ABB RAPID module: FrameFieldProbe.mod

MODULE FrameFieldProbe
    ! CrossArm - frame field probe: see tools/make_frame_field_probe.py.
    PERS tooldata ffStylus:=[TRUE,[[0,0,150],[1,0,0,0]],[3,[0,0,50],[1,0,0,0],0,0,0]];
    PERS wobjdata ffPallet:=[FALSE,TRUE,"",[[1000,0,800],[0,0,1,0]],[[0,0,0],[1,0,0,0]]];
    PERS wobjdata ffNest1:=[FALSE,TRUE,"",[[1000,0,800],[0,0,1,0]],[[0,0,0],[1,0,0,0]]];
    PERS wobjdata ffNest2:=[FALSE,TRUE,"",[[1000,0,800],[0,0,1,0]],[[0,0,0],[1,0,0,0]]];
    PERS wobjdata ffNest3:=[FALSE,TRUE,"",[[1000,0,800],[0,0,1,0]],[[0,0,0],[1,0,0,0]]];
    PERS wobjdata ffNest4:=[FALSE,TRUE,"",[[1000,0,800],[0,0,1,0]],[[0,0,0],[1,0,0,0]]];
    PERS wobjdata ffNest5:=[FALSE,TRUE,"",[[1000,0,800],[0,0,1,0]],[[0,0,0],[1,0,0,0]]];
    PERS wobjdata ffNest6:=[FALSE,TRUE,"",[[1000,0,800],[0,0,1,0]],[[0,0,0],[1,0,0,0]]];
    PERS wobjdata ffNest7:=[FALSE,TRUE,"",[[1000,0,800],[0,0,1,0]],[[0,0,0],[1,0,0,0]]];
    PERS wobjdata ffNest8:=[FALSE,TRUE,"",[[1000,0,800],[0,0,1,0]],[[30,0,0],[1,0,0,0]]];
    PERS wobjdata ffNest9:=[FALSE,TRUE,"",[[1000,0,800],[0,0,1,0]],[[0,20,0],[0.9659258,0,0,0.258819]]];
    CONST robtarget ffT1:=[[950,-60,820],[0,-0.1736482,0.9848078,0],[0,0,0,0],[9E9,9E9,9E9,9E9,9E9,9E9]];
    CONST robtarget ffT2:=[[1050,80,780],[0,0,1,0],[0,0,0,0],[9E9,9E9,9E9,9E9,9E9,9E9]];
    CONST robtarget ffTipNom:=[[0,0,150],[1,0,0,0],[0,0,0,0],[9E9,9E9,9E9,9E9,9E9,9E9]];
    CONST robtarget ffP:=[[40,30,-60],[1,0,0,0],[0,0,0,0],[9E9,9E9,9E9,9E9,9E9,9E9]];
    VAR robtarget ffM1;
    VAR robtarget ffM2;
    VAR robtarget ffOfs;
    VAR robtarget ffF1;
    VAR robtarget ffF2;
    VAR robtarget ffF3;
    VAR robtarget ffF4;
    VAR robtarget ffF5;
    VAR robtarget ffF6;
    VAR robtarget ffF7;
    VAR robtarget ffF8;
    VAR robtarget ffF9;
    VAR robtarget ffF10;
    VAR robtarget ffF11;
    VAR num ffDone:=0;

    PROC FfConv()
        ffDone:=0;
        MoveJ ffT2,v500,fine,tool0;
        ffM2:=CRobT(\Tool:=tool0\WObj:=wobj0);
        ffOfs:=Offs(ffTipNom,0,0,ffM2.trans.z-760);
        ffStylus.tframe.trans:=ffOfs.trans;
        ffStylus.tframe.trans.x:=ffM2.trans.x-1040;
        MoveL ffT2,v500,fine,ffStylus;
        ffF1:=CRobT(\Tool:=tool0\WObj:=wobj0);
        MoveJ ffT1,v500,fine,tool0;
        ffM1:=CRobT(\Tool:=tool0\WObj:=wobj0);
        ffPallet.uframe.trans:=ffM1.trans;
        ffPallet.uframe.rot:=ffM1.rot;
        ffPallet.oframe:=[[0,0,0],[1,0,0,0]];
        MoveL ffP,v500,fine,tool0\WObj:=ffPallet;
        ffF2:=CRobT(\Tool:=tool0\WObj:=wobj0);
        ffNest1.uframe:=ffPallet.uframe;
        ffNest3.uframe:=ffPallet.uframe;
        ffNest4.uframe:=ffPallet.uframe;
        ffNest5.uframe:=ffPallet.uframe;
        ffNest6.uframe:=ffPallet.uframe;
        ffNest7.uframe:=ffPallet.uframe;
        ffNest8.uframe:=ffPallet.uframe;
        ffNest9.uframe:=ffPallet.uframe;
        ffNest2.uframe:=[ffM2.trans,ffPallet.uframe.rot];
        MoveL ffP,v500,fine,tool0\WObj:=ffNest1;
        ffF3:=CRobT(\Tool:=tool0\WObj:=wobj0);
        MoveL ffP,v500,fine,tool0\WObj:=ffNest8;
        ffF4:=CRobT(\Tool:=tool0\WObj:=wobj0);
        MoveL ffP,v500,fine,tool0\WObj:=ffNest9;
        ffF5:=CRobT(\Tool:=tool0\WObj:=wobj0);
        MoveL ffP,v500,fine,tool0\WObj:=ffNest2;
        ffF6:=CRobT(\Tool:=tool0\WObj:=wobj0);
        MoveL ffP,v500,fine,tool0\WObj:=ffNest3;
        ffF7:=CRobT(\Tool:=tool0\WObj:=wobj0);
        MoveL ffP,v500,fine,tool0\WObj:=ffNest4;
        ffF8:=CRobT(\Tool:=tool0\WObj:=wobj0);
        MoveL ffP,v500,fine,tool0\WObj:=ffNest5;
        ffF9:=CRobT(\Tool:=tool0\WObj:=wobj0);
        MoveL ffP,v500,fine,tool0\WObj:=ffNest6;
        ffF10:=CRobT(\Tool:=tool0\WObj:=wobj0);
        MoveL ffP,v500,fine,tool0\WObj:=ffNest7;
        ffF11:=CRobT(\Tool:=tool0\WObj:=wobj0);
        ffDone:=1;
    ENDPROC
ENDMODULE
